PROGRAM POU
VAR
	pointer1 : POINTER TO DATE_AND_TIME := ADR(GVL.TimeDateInit);
	reference1 : REFERENCE TO TIME REF= GVL.TimeInit;
END_VAR

pointer1^ := DT#2024-2-8-14:51:0;
reference1 := TIME#4000ms;

END_PROGRAM

(* stored: Version 1.1.0.1, ProductVersion 3.1.4024.12
   POU POU: Id {99c0f409-0535-4753-b519-30628b42ccf3}, SpecialFunc None *)
